TYPE stRecMan_ListEntry :
STRUCT
	sFileName:STRING;
	dtCreationTime:DT;
END_STRUCT
END_TYPE

(* stored: Version 1.1.0.1, ProductVersion 3.1.4024.4
   DUT stRecMan_ListEntry: Id {685e9c86-a0f2-4dbe-a669-012386636ccf} *)
